FUNCTION_BLOCK Counter
VAR_INPUT
	
END_VAR
VAR_OUTPUT
	timeElapsed: TIME := T#0S;
END_VAR
VAR
	readyToCount : BOOL := FALSE;
	timeStart: TIME;  
 	timerRunning: BOOL := FALSE;
	//timeOne : TIME;
END_VAR


IF GVL.sensorN1 AND GVL.sensorN2 THEN
	readyToCount := TRUE;
END_IF

IF NOT GVL.sensorN1 AND readyToCount THEN
	timeStart := TIME();
	readyToCount := FALSE;
	timerRunning := TRUE;
END_IF

IF NOT GVL.sensorN2 AND timerRunning THEN
	timeElapsed := TIME() - timeStart;
	timerRunning := FALSE;
END_IF





(* IF startMeasurement AND NOT GVL.sensorN1 THEN
    timerRunning := TRUE;
    timeStart := TIME();
	timeOne := timeStart;
	startMeasurement := FALSE;
END_IF

IF timerRunning AND NOT GVL.sensorN2 THEN
    timeElapsed := TIME() - timeOne;
    timerRunning := FALSE;
END_IF *)

END_FUNCTION_BLOCK

(* stored: Version 1.1.0.1, ProductVersion 3.1.4024.13
   POU Counter: Id {fc193301-d8f2-4dd8-aee4-498ebab1a227}, SpecialFunc None *)
